FUNCTION_BLOCK Seq_Get_Plate EXTENDS FB_BASIS IMPLEMENTS I_Sequenz
VAR_INPUT
	// Benötigte Skills
	Move_Robot			:I_Skill_Roboter;
	Move_Gripper		:I_Skill_Greifer; 
	
	// Benötigte Parameter
	R_Plate_Pos			:sRoboterProzessVariablen; 
	R_Offset			:LREAL;
	
	G_Ready_Pos			:sSmartGreiferProzessVariablen;
	G_Grip_Pos			:sSmartGreiferProzessVariablen;
	
END_VAR

VAR_OUTPUT
END_VAR

VAR
	R_Offset_Pos		:sRoboterProzessVariablen; 
END_VAR

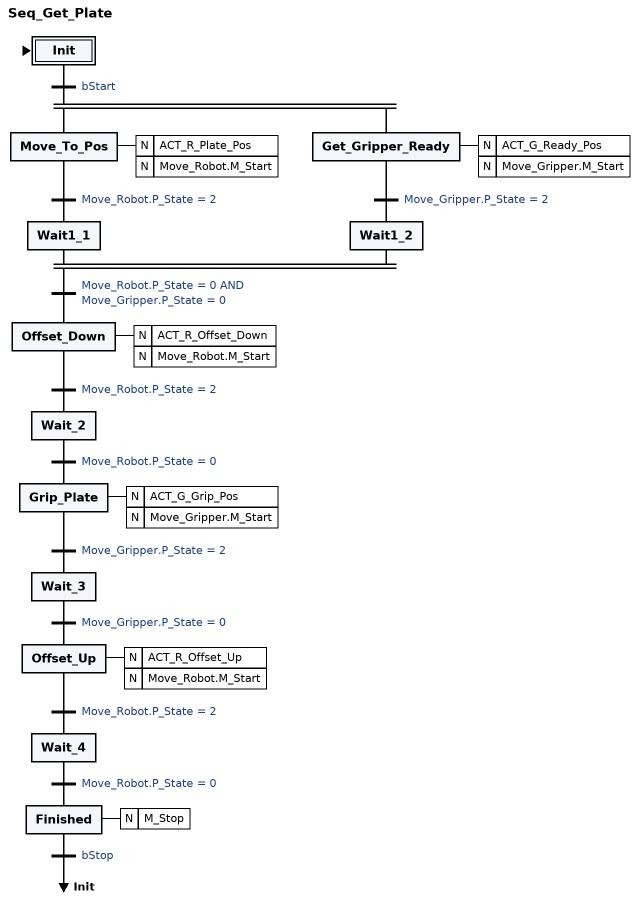
INITIAL_STEP Init:
END_STEP
TRANSITION FROM Init TO (Move_To_Pos, Get_Gripper_Ready)
    := bStart;
END_TRANSITION
STEP Move_To_Pos:
    ACT_R_Plate_Pos(N);
    Move_Robot.M_Start(N);
END_STEP
TRANSITION FROM Move_To_Pos TO Wait1_1
    := Move_Robot.P_State = 2;
END_TRANSITION
STEP Wait1_1:
END_STEP
STEP Get_Gripper_Ready:
    ACT_G_Ready_Pos(N);
    Move_Gripper.M_Start(N);
END_STEP
TRANSITION FROM Get_Gripper_Ready TO Wait1_2
    := Move_Gripper.P_State = 2;
END_TRANSITION
STEP Wait1_2:
END_STEP
TRANSITION FROM (Wait1_1, Wait1_2) TO Offset_Down
    := Move_Robot.P_State = 0 AND Move_Gripper.P_State = 0;
END_TRANSITION
STEP Offset_Down:
    ACT_R_Offset_Down(N);
    Move_Robot.M_Start(N);
END_STEP
TRANSITION FROM Offset_Down TO Wait_2
    := Move_Robot.P_State = 2;
END_TRANSITION
STEP Wait_2:
END_STEP
TRANSITION FROM Wait_2 TO Grip_Plate
    := Move_Robot.P_State = 0;
END_TRANSITION
STEP Grip_Plate:
    ACT_G_Grip_Pos(N);
    Move_Gripper.M_Start(N);
END_STEP
TRANSITION FROM Grip_Plate TO Wait_3
    := Move_Gripper.P_State = 2;
END_TRANSITION
STEP Wait_3:
END_STEP
TRANSITION FROM Wait_3 TO Offset_Up
    := Move_Gripper.P_State = 0;
END_TRANSITION
STEP Offset_Up:
    ACT_R_Offset_Up(N);
    Move_Robot.M_Start(N);
END_STEP
TRANSITION FROM Offset_Up TO Wait_4
    := Move_Robot.P_State = 2;
END_TRANSITION
STEP Wait_4:
END_STEP
TRANSITION FROM Wait_4 TO Finished
    := Move_Robot.P_State = 0;
END_TRANSITION
STEP Finished:
    M_Stop(N);
END_STEP
TRANSITION FROM Finished TO Init
    := bStop;
END_TRANSITION

ACTION ACT_G_Grip_Pos:
Move_Gripper.P_Prozessparameter := G_Grip_Pos;
END_ACTION

ACTION ACT_G_Ready_Pos:
Move_Gripper.P_Prozessparameter := G_Ready_Pos;
END_ACTION

ACTION ACT_R_Offset_Down:
R_Offset_Pos.q3 := -R_Offset;
R_Offset_Pos.v := 0.1;
R_Offset_Pos.a := 0.1;
R_Offset_Pos.MoveTyp := 0;
R_Offset_Pos.PosTyp := 1;

Move_Robot.P_Prozessparameter := R_Offset_Pos;
END_ACTION

ACTION ACT_R_Offset_Up:
R_Offset_Pos.q3 := R_Offset;
R_Offset_Pos.v := 0.2;
R_Offset_Pos.a := 0.2;
R_Offset_Pos.MoveTyp := 0;
R_Offset_Pos.PosTyp := 1;

Move_Robot.P_Prozessparameter := R_Offset_Pos;
END_ACTION

ACTION ACT_R_Plate_Pos:
Move_Robot.P_Prozessparameter := R_Plate_Pos;
END_ACTION

END_FUNCTION_BLOCK

(* stored: Version 1.1.0.1
   POU Seq_Get_Plate: Id {3c2f7a5d-847d-4bf0-bae9-2120fa4adec2}, SpecialFunc None
   Folder 01_Zuweisung: Id {a28adf77-c645-4ef1-9290-4d6a3b107eae}
   Action ACT_G_Grip_Pos: Id {701b0338-d740-48ac-83e5-4ad64166a15d}
   Action ACT_G_Ready_Pos: Id {ec9bbaae-8df0-4b3a-a5fc-597168e2fef6}
   Action ACT_R_Offset_Down: Id {093c7b63-c93a-4f1c-b8b0-68c41266a1e5}
   Action ACT_R_Offset_Up: Id {e61199a1-77cd-4d54-95f2-4d3b407512b5}
   Action ACT_R_Plate_Pos: Id {914fa552-e92b-4e3c-b7c6-dcca0102578f} *)
